// LS Electric XG5000 project: 0131 인버터 다단속
// PLC LSPLC

PROGRAM NewProgram (task: 스캔 프로그램)

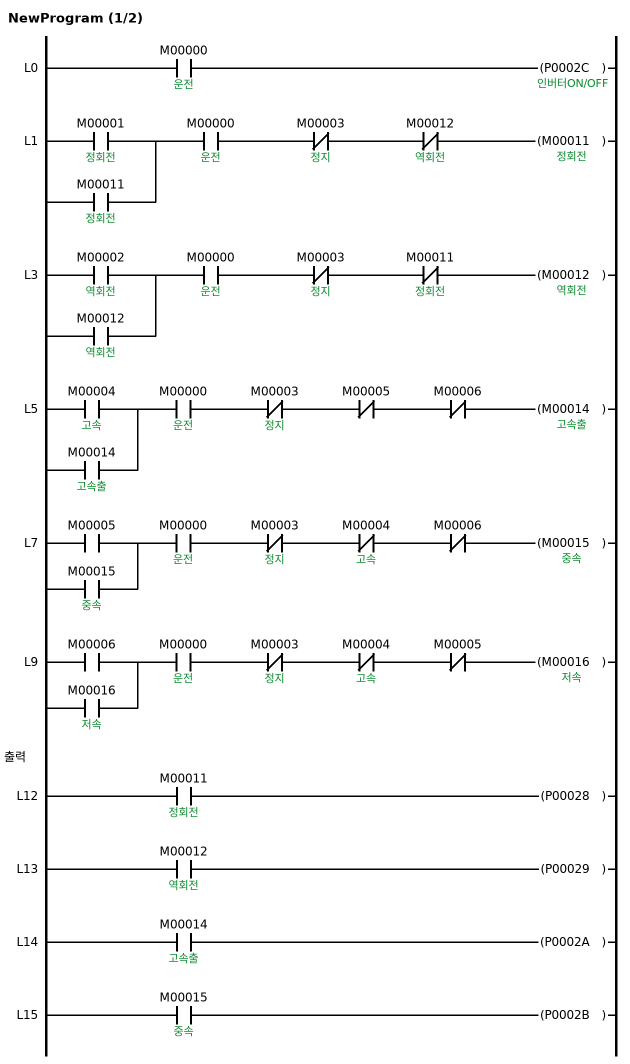
; L0
LOAD      M00000	// 운전
OUT       P0002C	// 인버터ON/OFF
; L1
LOAD      M00001	// 정회전
OR        M00011	// 정회전
AND       M00000	// 운전
AND NOT   M00003	// 정지
AND NOT   M00012	// 역회전
OUT       M00011	// 정회전
; L3
LOAD      M00002	// 역회전
OR        M00012	// 역회전
AND       M00000	// 운전
AND NOT   M00003	// 정지
AND NOT   M00011	// 정회전
OUT       M00012	// 역회전
; L5
LOAD      M00004	// 고속
OR        M00014	// 고속출
AND       M00000	// 운전
AND NOT   M00003	// 정지
AND NOT   M00005
AND NOT   M00006
OUT       M00014	// 고속출
; L7
LOAD      M00005
OR        M00015	// 중속
AND       M00000	// 운전
AND NOT   M00003	// 정지
AND NOT   M00004	// 고속
AND NOT   M00006
OUT       M00015	// 중속
; L9
LOAD      M00006
OR        M00016	// 저속
AND       M00000	// 운전
AND NOT   M00003	// 정지
AND NOT   M00004	// 고속
AND NOT   M00005
OUT       M00016	// 저속
출력:
; L12
LOAD      M00011	// 정회전
OUT       P00028
; L13
LOAD      M00012	// 역회전
OUT       P00029
; L14
LOAD      M00014	// 고속출
OUT       P0002A
; L15
LOAD      M00015	// 중속
OUT       P0002B

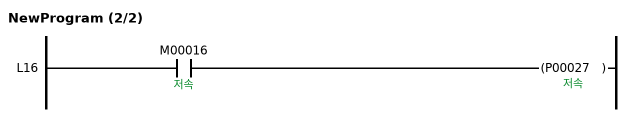
; L16
LOAD      M00016	// 저속
OUT       P00027	// 저속

VARIABLES AND COMMENTS (devices not used above)
P00004	BIT	중속
P00006	BIT	출구
P00003	BIT	고속